PROGRAM Axis_2
VAR
	bLimitPowerAxis2 AT %Q*: BOOL := TRUE;
END_VAR

//Initial parameters of an Axis
IF _TaskInfo[fbGetCurTaskIndex.index].FirstCycle THEN
    //Initial default values:
    GVL.astAxes[2].stConfig.eHomeSeq := 1;
    GVL.astAxes[2].stConfig.fHomePosition := 0.0;
    GVL.astAxes[2].stConfig.fHomeFinishDistance := -1;
END_IF

//Define ACTIONS() or write exclusive code for an specific axis.
//Eg. Stop when temperature reaches certain values, reduce speed if  a signal is activated, etc.

ACT_2_Interlock();

// Brake control from GUI
main.stHWControlY.bBrakeReleaseCmd:=main.stCmdEpics.bYReleaseBreakCmd;
main.stHWStatusY.bBrakeReleased:=main.stHWControlY.bBrakeReleaseCmd;

ACTION ACT_2_Interlock:
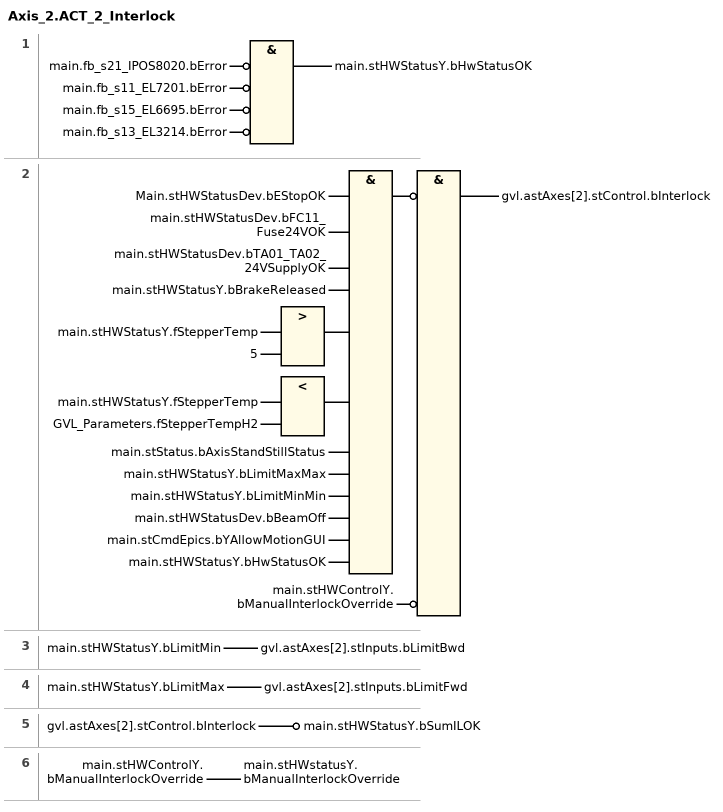
// NETWORK 1
main.stHWStatusY.bHwStatusOK := NOT main.fb_s21_IPOS8020.bError AND NOT main.fb_s11_EL7201.bError AND NOT main.fb_s15_EL6695.bError AND NOT main.fb_s13_EL3214.bError;

// NETWORK 2
gvl.astAxes[2].stControl.bInterlock := NOT (Main.stHWStatusDev.bEStopOK AND main.stHWStatusDev.bFC11_Fuse24VOK AND main.stHWStatusDev.bTA01_TA02_24VSupplyOK AND main.stHWStatusY.bBrakeReleased AND main.stHWStatusY.fStepperTemp > 5 AND main.stHWStatusY.fStepperTemp < GVL_Parameters.fStepperTempH2 AND main.stStatus.bAxisStandStillStatus AND main.stHWStatusY.bLimitMaxMax AND main.stHWStatusY.bLimitMinMin AND main.stHWStatusDev.bBeamOff AND main.stCmdEpics.bYAllowMotionGUI AND main.stHWStatusY.bHwStatusOK) AND NOT main.stHWControlY.bManualInterlockOverride;

// NETWORK 3
gvl.astAxes[2].stInputs.bLimitBwd := main.stHWStatusY.bLimitMin;

// NETWORK 4
gvl.astAxes[2].stInputs.bLimitFwd := main.stHWStatusY.bLimitMax;

// NETWORK 5
main.stHWStatusY.bSumILOK := NOT gvl.astAxes[2].stControl.bInterlock;

// NETWORK 6
main.stHWstatusY.bManualInterlockOverride := main.stHWControlY.bManualInterlockOverride;
END_ACTION

END_PROGRAM

(* stored: Version 1.1.0.1, ProductVersion 3.1.4024.6
   POU Axis_2: Id {cc52a494-82bc-4d82-99c3-9bfba67cd4d8}, SpecialFunc None
   Action ACT_2_Interlock: Id {c949121c-9701-4c5f-8bc8-3c78316b1a11} *)
